TYPE enum_E:
    (elit_BlinkQ1Off, elit_BlinkQ1On, elit_init0, elit_init1, elit_init2, elit_init_error, elit_init_ok, elit_init_sensor_check, elit_initialized, elit_Off, elit_On, elit_Q2Activated, elit_Start, elit_Wait2s, elit_WaitForRelease);
END_TYPE

(* stored: ProductVersion 3.1.0.18, Version 1.1.0.1 *)
